// TIA Portal project "3M-2" (V16)

(* hardware
DEVICE "S7-1200 station_1"  S7-1200 Station
   slot 0: "Rack_0"  S7-1200 Rack  Rack  V1.0
   slot 1: "PLC_1"  CPU 1212C AC/DC/Rly  6ES7 212-1BE40-0XB0  V4.0
*)

// ===== PLC "PLC_1"  CPU 1212C AC/DC/Rly =====

VAR_GLOBAL   // PLC tag table "Default tag table"
   "K1" AT %Q0.0 : Bool;
   "stop1" AT %I0.4 : Bool;
   "k2" AT %Q0.1 : Bool;
   "X" AT %M0.0 : Bool;
   "K3" AT %Q0.2 : Bool;
   "start1" AT %I0.2 : Bool;
   "T1 tag" AT %M0.1 : Bool;
   "T2 tag" AT %M0.2 : Bool;
   "T3 tag" AT %M0.3 : Bool;
   "Y" AT %M1.0 : Bool;
   "T4 tag" AT %M1.2 : Bool;
   "Tag_1" AT %M1.1 : Bool;
   "T5 tag" AT %M1.3 : Bool;
   "Tag_2" AT %M1.6 : Bool;
END_VAR

// folder: System blocks/Program resources

DATA_BLOCK "T4"   // DB1
{ S7_Optimized_Access := 'TRUE' }
AUTHOR : Simatic
FAMILY : IEC
NAME : IEC_TMR
VERSION : 1.0
// stored: InstanceOfName IEC_TIMER
"IEC_TIMER"
BEGIN
END_DATA_BLOCK

DATA_BLOCK "T1"   // DB2
{ S7_Optimized_Access := 'TRUE' }
AUTHOR : Simatic
FAMILY : IEC
NAME : IEC_TMR
VERSION : 1.0
// stored: InstanceOfName IEC_TIMER
"IEC_TIMER"
BEGIN
END_DATA_BLOCK

DATA_BLOCK "T2"   // DB3
{ S7_Optimized_Access := 'TRUE' }
AUTHOR : Simatic
FAMILY : IEC
NAME : IEC_TMR
VERSION : 1.0
// stored: InstanceOfName IEC_TIMER
"IEC_TIMER"
BEGIN
END_DATA_BLOCK

DATA_BLOCK "T3"   // DB4
{ S7_Optimized_Access := 'TRUE' }
AUTHOR : Simatic
FAMILY : IEC
NAME : IEC_TMR
VERSION : 1.0
// stored: InstanceOfName IEC_TIMER
"IEC_TIMER"
BEGIN
END_DATA_BLOCK

DATA_BLOCK "T5"   // DB5
{ S7_Optimized_Access := 'TRUE' }
AUTHOR : Simatic
FAMILY : IEC
NAME : IEC_TMR
VERSION : 1.0
// stored: InstanceOfName IEC_TIMER
"IEC_TIMER"
BEGIN
END_DATA_BLOCK

// folder: (top level)

ORGANIZATION_BLOCK "Main"   // OB1, LAD, ProgramCycle
TITLE = "Main Program Sweep (Cycle)"
{ S7_Optimized_Access := 'TRUE' }
VERSION : 0.1
   VAR_INPUT
      Initial_Call : Bool;   // Initial call of this OB
      Remanence : Bool;   // =True, if remanent data are available
   END_VAR
BEGIN

REGION Network 1: start
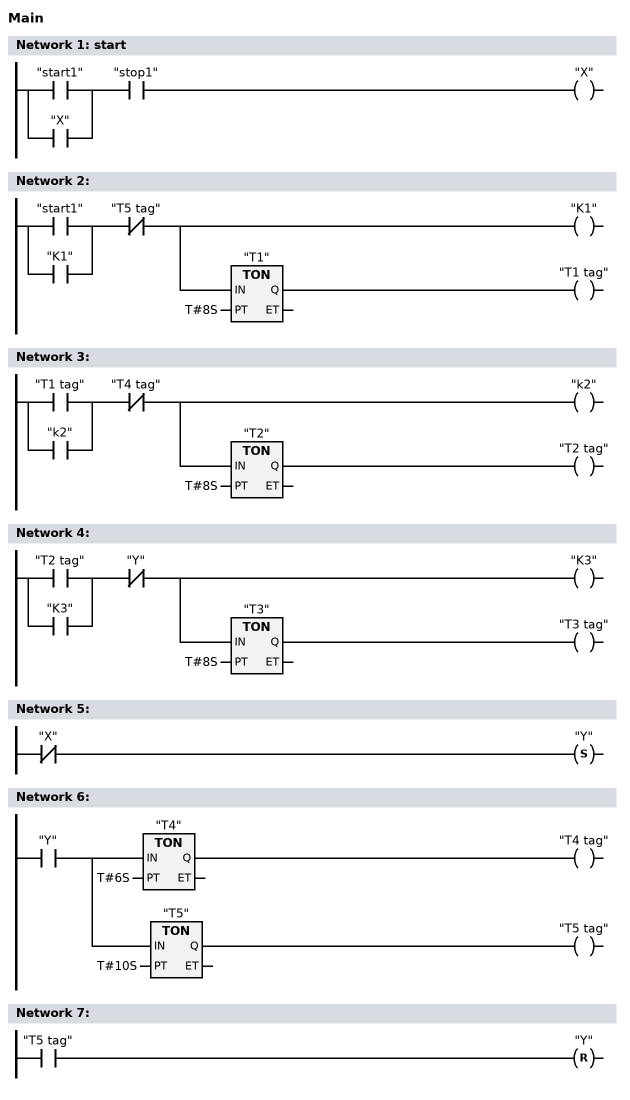
   RUNG wire#powerrail
      Contact( "start1" )
      wire#w1
      Contact( "stop1" )
      Coil( "X" )
   END_RUNG
   RUNG wire#powerrail
      Contact( "X" )
   END_RUNG wire#w1
   // the same network as SCL:
   "X" := ("start1" OR "X") AND "stop1";
END_REGION

REGION Network 2
   "K1" := ("start1" OR "K1") AND NOT "T5 tag";
   "T1".TON(IN := "K1", PT := T#8S);
   "T1 tag" := "T1".Q;
END_REGION

REGION Network 3
   "k2" := ("T1 tag" OR "k2") AND NOT "T4 tag";
   "T2".TON(IN := "k2", PT := T#8S);
   "T2 tag" := "T2".Q;
END_REGION

REGION Network 4
   "K3" := ("T2 tag" OR "K3") AND NOT "Y";
   "T3".TON(IN := "K3", PT := T#8S);
   "T3 tag" := "T3".Q;
END_REGION

REGION Network 5
   RUNG wire#powerrail
      I_Contact( "X" )
      S_Coil( "Y" )
   END_RUNG
   // the same network as SCL:
   IF NOT "X" THEN "Y" := TRUE; END_IF;
END_REGION

REGION Network 6
   "T4".TON(IN := "Y", PT := T#6S);
   "T4 tag" := "T4".Q;
   "T5".TON(IN := "Y", PT := T#10S);
   "T5 tag" := "T5".Q;
END_REGION

REGION Network 7
   RUNG wire#powerrail
      Contact( "T5 tag" )
      R_Coil( "Y" )
   END_RUNG
   // the same network as SCL:
   IF "T5 tag" THEN "Y" := FALSE; END_IF;
END_REGION
END_ORGANIZATION_BLOCK